FUNCTION Call_OperatingMode

instOperatingMode(PermissionHardware:= simPermissionHardware, 
				  PermissionSoftware:= simPermissionSafety, 
				  E_Stop:= E_Stop, 
				  OperatingModeManual:= BetrMan, 
				  OperatingModeAutomatic:= BetrAuto, 
				  LEDStart=> StartLED, 
				  LEDStop=> StopLED, 
				  LEDHome=> HomeLED, 
				  LEDReset=> ResetLED, 
				  LEDQuit=> QuitLED);

instOperatingMode.Start_On(StartButton);
instOperatingMode.Stop_On(StopButton);
instOperatingMode.Homeing_On(HomeButton);
instOperatingMode.Reset_On(ResetButton);
instOperatingMode.Quit_On(QuitButton);

END_FUNCTION

(* stored: Version 1.1.0.1
   POU Call_OperatingMode: Id {e0abeec7-2c06-4fbb-ba98-ebafc89ce1b0}, SpecialFunc None *)
